{attribute 'TcGenerated'}
// This function has been automatically generated from the project information.
VAR_GLOBAL CONSTANT
    {attribute 'const_non_replaced'}
    {attribute 'linkalways'}
    stLibVersion_lcls_plc_crix_motion : ST_LibVersion := (iMajor := 1, iMinor := 2, iBuild := 0, iRevision := 0, sVersion := '1.2.0');
END_VAR

(* stored: Version 1.1.0.1, ProductVersion 3.1.4022.18
   GVL Global_Version: Id a605e153-0b6e-4f2f-8928-f647432e2442 *)
